// TwinCAT 3 PLC project Marquee
// Title: Marquee
// Company: HiJack Automation
// ProjectVersion: 0.5
// Description: fix bug->press Stop button, then all lamp OFF 0.5: fix bug-> press start button can re-start the Rolling cycle
// ProgramVersion: 3.1.4022.4
// libraries:
//   Tc2_Standard, * (Beckhoff Automation GmbH)
//   Tc2_System, * (Beckhoff Automation GmbH)
//   Tc3_Module, * (Beckhoff Automation GmbH)
// project tree:
//   FBs/ FB_Marquee.TcPOU, FB_MarqueeEx.TcPOU, FB_MarqueeExPause.TcPOU
//   / PlcTask.TcTTO
//   POUs/ MAIN.TcPOU
// real-time tasks:
//   TASK PlcTask: cycle T#10ms, priority 20, ADS port 350

CONFIGURATION Marquee
    RESOURCE PLC ON TwinCAT3
        TASK PlcTask(INTERVAL := T#10ms, PRIORITY := 20);
        PROGRAM MAIN WITH PlcTask : MAIN;
    END_RESOURCE
END_CONFIGURATION

// ---- POUs/MAIN.TcPOU
PROGRAM MAIN
VAR
	(*fbMarquee		:FB_Marquee;
	bLamp01,bLamp02,bLamp03,bLamp04		:BOOL;
	bBlinking			:BOOL;
	
	fbMarqueeEx		:FB_MarqueeEx;
	tDelay			:TIME:=T#500MS;
	
	
	fbMarqueeExPause		:FB_MarqueeExPause;
	bPause					:BOOL;
	bStop					:BOOL;  *)
END_VAR

//==========Test FB_Marquee===========
//fbMarquee(pLamp01:= ADR(bLamp01) , pLamp02:=ADR(bLamp02), pLamp03:=ADR(bLamp03) , pLamp04:= ADR(bLamp04));
//fbMarquee.Blinking(bStart :=bBlinking );
//==========Test FB_Marquee===========


//===============Test FB_MarqueeEx======================
//fbMarqueeEx(pLamp01:= ADR(bLamp01) , pLamp02:=ADR(bLamp02),
//			 pLamp03:=ADR(bLamp03) , pLamp04:= ADR(bLamp04),pTime:= ADR(tDelay));
			 
//fbMarqueeEx.Blinking(bStart := bBlinking);
//===============Test FB_MarqueeEx======================


//===============Test FB_MarqueeExPause======================
(*fbMarqueeExPause(pLamp01:= ADR(bLamp01) , pLamp02:=ADR(bLamp02),
			 pLamp03:=ADR(bLamp03) , pLamp04:= ADR(bLamp04),pTime:= ADR(tDelay),pPause:= ADR(bPause),pStop := ADR(bStop));
fbMarqueeExPause.Blinking(bStart :=bBlinking);  *)

END_PROGRAM

// ---- FBs/FB_Marquee.TcPOU
FUNCTION_BLOCK FB_Marquee
//trigger all four light rolling on and off one by one loop. On for 1 second.
VAR_INPUT
	pLamp01			:POINTER TO BOOL;
	pLamp02			:POINTER TO BOOL;
	pLamp03			:POINTER TO BOOL;
	pLamp04			:POINTER TO BOOL;
END_VAR
VAR_OUTPUT
END_VAR
VAR
	TON1		:TON;	
	iStep		:INT;	
END_VAR

METHOD Blinking : BOOL
VAR_INPUT
	bStart			:BOOL;
END_VAR
VAR
	
END_VAR
(*IF bStart THEN
	 
	TON1(IN:=TRUE, PT:= T#1S, Q=> , ET=> );
	pLamp01^ := TRUE;
	
	IF	TON1.Q THEN 
		pLamp01^ := FALSE;
		TON2(IN:=TON1.Q, PT:= T#1S, Q=> , ET=> );
		pLamp02^ := TRUE;
		IF TON2.Q THEN 
			pLamp02^ := FALSE;
			TON3(IN:=TON2.Q, PT:= T#1S, Q=> , ET=> );
			pLamp03^ := TRUE;
			IF TON3.Q THEN 
				pLamp03^ := FALSE;
				TON4(IN:=TON3.Q, PT:= T#1S, Q=> , ET=> );
				pLamp04^ := TRUE;
				IF TON4.Q THEN 
					pLamp04^ := FALSE;
					TON1(IN:=FALSE);
					
				END_IF
			END_IF
		END_IF
	END_IF *)
	
IF bStart THEN 
	CASE iStep OF
			0:
				pLamp01^ := TRUE;
				TON1(IN:=TRUE, PT:= T#1S, Q=> , ET=> );
				IF TON1.Q THEN 
					pLamp01^ := FALSE;
					TON1(IN:=FALSE);
					iStep:= 10;
				END_IF				
			10:
				pLamp02^ := TRUE;
				TON1(IN:=TRUE, PT:=T#1S, Q=> , ET=> );
				IF TON1.Q THEN 
					pLamp02^ := FALSE;
					TON1(IN:=FALSE);
					iStep := 20;				
				END_IF
			20:
				pLamp03^ := TRUE;
				TON1(IN:=TRUE, PT:=T#1S, Q=> , ET=> );
				IF TON1.Q THEN 
					pLamp03^ := FALSE;
					TON1(IN:=FALSE);
					iStep := 30;
				END_IF
			30:
				pLamp04^ := TRUE;
				TON1(IN:=TRUE, PT:=T#1S, Q=> , ET=> );
				IF	TON1.Q THEN 
					pLamp04^ := NOT pLamp04^;
					TON1(IN:=FALSE);
					iStep := 0;
				END_IF
	END_CASE
ELSE 
	pLamp04^ := FALSE;
	pLamp03^ := FALSE;
	pLamp02^ := FALSE;
	pLamp01^ := FALSE;
END_IF
END_METHOD

END_FUNCTION_BLOCK

// ---- FBs/FB_MarqueeEx.TcPOU
FUNCTION_BLOCK FB_MarqueeEx EXTENDS FB_Marquee
//trigger all four light rolling on and off one by one loop. Ptime is the On elapse time
VAR_INPUT	
	pTime		:POINTER TO TIME;
END_VAR
VAR_OUTPUT
END_VAR
VAR
	bDelayOK		:BOOL;
	iDelayStep		:UDINT;
END_VAR

METHOD Blinking : BOOL
VAR_INPUT
	bStart			:BOOL;
END_VAR
VAR
	
END_VAR
IF bStart THEN 
	CASE iStep OF 
		0:
			pLamp01^ := TRUE;
			THIS^.Delay();
			IF THIS^.bDelayOK THEN 
				pLamp01^ := NOT pLamp01^;
				THIS^.Reset();
				iStep := 10;
			END_IF
		10:
			pLamp02^ := TRUE;
			THIS^.Delay();
			IF bDelayOK THEN 
				pLamp02^ := NOT pLamp02^;
				THIS^.Reset();
				iStep := 20;
			END_IF
		20:
			pLamp03^ := TRUE;
			THIS^.Delay();
			IF bDelayOK THEN 
				pLamp03^ := NOT pLamp03^;
				THIS^.Reset();
				iStep := 30;
			END_IF
		30:
			pLamp04^ := TRUE;
			THIS^.Delay();
			IF bDelayOK THEN 
				pLamp04^ := NOT pLamp04^;
				THIS^.Reset();
				iStep := 0;
			END_IF		
	END_CASE
ELSE 
	pLamp04^ := FALSE;
	pLamp03^ := FALSE;
	pLamp02^ := FALSE;
	pLamp01^ := FALSE;
END_IF
END_METHOD

METHOD Delay : BOOL
VAR_INPUT
END_VAR
CASE iDelayStep OF
	0:
		bDelayOK := FALSE;
		TON1(IN:=FALSE);
		iDelayStep := 10;
	10:
		TON1(IN:=TRUE , PT:= pTime^, Q=> , ET=> );
		IF TON1.Q THEN 
			TON1(IN:=FALSE);
			bDelayOK := TRUE;
			iDelayStep := 100;
		END_IF
END_CASE
END_METHOD

METHOD Reset : BOOL
VAR_INPUT
END_VAR
iDelayStep := 0;
bDelayOK := FALSE;

TON1(IN:=FALSE);
END_METHOD

END_FUNCTION_BLOCK

// ---- FBs/FB_MarqueeExPause.TcPOU
FUNCTION_BLOCK FB_MarqueeExPause EXTENDS FB_MarqueeEx
VAR_INPUT
	pPause		:POINTER TO BOOL;
	pStop		:POINTER TO BOOL;
END_VAR
VAR_OUTPUT
END_VAR
VAR
END_VAR

METHOD Blinking : BOOL
VAR_INPUT
	bStart			:BOOL;
END_VAR
VAR
	bRunning		:BOOL;
	fTrig		:F_TRIG;
END_VAR
IF bStart THEN	
	CASE iStep OF			
		0:
			bRunning := TRUE;
			pLamp01^ := TRUE;
			THIS^.Delay();
			IF THIS^.bDelayOK THEN 
				pLamp01^ := NOT pLamp01^;
				SUPER^.Reset();
				iStep := 10;
			END_IF
		10:
			pLamp02^ := TRUE;
			THIS^.Delay();
			IF bDelayOK THEN 
				pLamp02^ := NOT pLamp02^;
				SUPER^.Reset();
				iStep := 20;
			END_IF
		20:
			pLamp03^ := TRUE;
			THIS^.Delay();
			IF bDelayOK THEN 
				pLamp03^ := NOT pLamp03^;
				SUPER^.Reset();
				iStep := 30;
			END_IF
		30:
			pLamp04^ := TRUE;
			THIS^.Delay();
			IF bDelayOK THEN 
				pLamp04^ := FALSE;
				SUPER^.Reset();
				IF pStop^ THEN									
					iStep:= 40;
				ELSE
					iStep := 0;
				END_IF				
			END_IF	
		40:		
			pLamp04^ := FALSE;
			pLamp03^ := FALSE;
			pLamp02^ := FALSE;
			pLamp01^ := FALSE;				
			iStep := 50;
		50:			
			IF NOT pStop^ THEN 
				iStep := 0;
			END_IF			
	END_CASE
ELSE 
	pLamp04^ := FALSE;
	pLamp03^ := FALSE;
	pLamp02^ := FALSE;
	pLamp01^ := FALSE;
END_IF
END_METHOD

METHOD Delay : BOOL
VAR_INPUT
END_VAR
CASE iDelayStep OF
	0:
		bDelayOK := FALSE;
		TON1(IN:=FALSE);		 
		iDelayStep := 10;
	10:
		TON1(IN:=TRUE , PT:= pTime^, Q=> , ET=> );
		IF TON1.Q THEN 						
			IF NOT pPause^  THEN
				TON1(IN:=FALSE);
				bDelayOK := TRUE;
				iDelayStep := 100;
			END_IF
			
		END_IF
END_CASE
END_METHOD

METHOD Reset : BOOL
VAR_INPUT
END_VAR
SUPER^.Reset();
iStep := 0;
END_METHOD

END_FUNCTION_BLOCK
